(* IEC 61131-3 sources: ConveyorControl-with-PLC/4E_Gruppe1_Graf_Projekt1_HMI/Class/KeyPadAnum, 1 file *)

(* ---- KeyPadAnum.st ---- *)
(*!
<Class
	Name               = "KeyPadAnum"
	Revision           = "0.6"
	RealtimeTask       = "false"
	CyclicTask         = "false"
	BackgroundTask     = "false"
	Sigmatek           = "true"
	OSInterface        = "false"
	HighPriority       = "false"
	Automatic          = "false"
	UpdateMode         = "Prescan"
	IconPath           = ".\Class\KeyPadAnum\KeyPad.ico"
	SharedCommandTable = "true"
	Objectsize         = "(284,120)"
	Comment            = "class is used to get defaultimplementation of QWERTZ, QWERTY, AZERTY keyboard.&#13;&#10;keyboard differs on different languages&#13;&#10;set client &quot;Ima&quot; to IMA_WINDOW&#13;&#10;set client &quot;No&quot; to _WIN_EDITOR_ANUMERIC">
	<Channels>
		<Client Name="AltGr" Required="false" Internal="false" DefValue="1" Comment="set client to 1 when use of AltGr-key is necessary&#13;&#10;on the other hand client has to be set to 0"/>
		<Client Name="CapitalLetter" Required="false" Internal="false" DefValue="0" Comment="set client to 1 if capital letters are used without activated shift mode&#13;&#10;on the other hand set 0 to get capital letters when shift mode is activated"/>
		<Client Name="KeyPadImg" Required="true" Internal="true"/>
	</Channels>
	<RevDoku>
		<Owner Company="sigmatek" Author="kolott"/>
		<Dokumentation Revision="0.6" Date="2015-11-06" Author="kolott" Company="sigmatek" Description="sa32226, color of titlebar will work at several frames"/>
		<Dokumentation Revision="0.5" Date="2015-08-21" Author="kolott" Company="sigmatek" Description="betterment when using different frames"/>
		<Dokumentation Revision="0.4" Date="2014-02-07" Author="kolott" Company="sigmatek" Description="innovation titlelinepositioning"/>
		<Dokumentation Revision="0.3" Date="2013-10-02" Author="kolott" Company="sigmatek" Description="russian, ukrainian and greek keypad added"/>
		<Dokumentation Revision="0.1" Date="2013-07-10" Author="kolott" Company="sigmatek" Description="AltGr and CapitalLetter clients added"/>
		<Dokumentation Revision="0.0" Date="2013-03-06" Author="kolott" Company="sigmatek" Description="release"/>
	</RevDoku>
	<Network Name="KeyPadAnum">
		<!-- List of Components in this network -->
		<Components>
			<Object
				Name       = "_base"
				Class      = "_Screen"
				Position   = "(218,120)"
				Visualized = "true">
				<Channels>
					<Server Name="Screen"/>
					<Client Name="ImA" Value="IMA_WINDOW"/>
					<Client Name="Lse"/>
					<Client Name="No" Value="_WIN_EDITOR_ANUMERIC"/>
				</Channels>
			</Object>
			<Object
				Name       = "KeyPadImg"
				Class      = "KeyPadImages"
				Position   = "(210,420)"
				Visualized = "false">
				<Channels>
					<Server Name="ClassSvr"/>
				</Channels>
			</Object>
		</Components>
		<Comments>
		</Comments>
		<!-- List of Connections in this network -->
		<Connections>
			<Connection Source="this.Screen" Destination="_base.Screen" Vertices="(690,210),(518,210),"/>
			<Connection Source="_base.Lse" Destination="this.Lse" Vertices="(218,210),(38,210),"/>
			<Connection Source="_base.No" Destination="this.No" Vertices="(218,270),(38,270),"/>
			<Connection Source="_base.ImA" Destination="this.ImA" Vertices="(218,330),(38,330),"/>
			<Connection Source="this.KeyPadImg" Destination="KeyPadImg.ClassSvr"/>
		</Connections>
		<!-- Headerfiles -->
		<Options>
		</Options>
	</Network>
</Class>
*)
#pragma using _Screen

KeyPadAnum : CLASS
: _Screen
  //Servers:
  //Clients:
	KeyPadImg 	: CltChCmd_KeyPadImages;
	AltGr 	: CltCh_DINT;
	CapitalLetter 	: CltCh_DINT;
  //Variables:
		KeyButton_XOff 	: INT;
		KeyButton_YOff 	: INT;
		KeyButton_Width 	: INT;
		KeyButton_Height 	: INT;
		DoneByProgram 	: BOOL;
		YOff 	: INT;
  //Functions:

	FUNCTION KeyPadAnum
		VAR_OUTPUT
			ret_code 	: ConfStates;
		END_VAR;

	FUNCTION VIRTUAL GLOBAL S_Start
		VAR_INPUT
			pic 	: ^void;
			firsttime 	: BOOL;
		END_VAR;

	FUNCTION VIRTUAL GLOBAL S_CreateNew
		VAR_INPUT
			psetup 	: ^_NEWSCREENPROP;
		END_VAR
		VAR_OUTPUT
			retcode 	: BOOL;
		END_VAR;

	FUNCTION TAB KeyTab_QUERTZ;

	FUNCTION TAB KeyTab_QUERTY;

	FUNCTION VIRTUAL SelectKeyboard
		VAR_OUTPUT
			retcode 	: ^USINT;
		END_VAR;

	FUNCTION TAB KeyTab_FRENCH;

	FUNCTION TAB KeyTab_ITALIAN;

	FUNCTION TAB KeyTab_SPAIN;

	FUNCTION TAB KeyTab_PORTUGUESE;

	FUNCTION TAB KeyTab_NORWEGIAN;

	FUNCTION TAB KeyTab_SWEDISH;

	FUNCTION TAB SingleText;

	FUNCTION VIRTUAL GetBig
		VAR_INPUT
			pkey 	: ^USINT;
		END_VAR
		VAR_OUTPUT
			retcode 	: USINT;
		END_VAR;

	FUNCTION TAB KeyTab_CROATIAN_SERBIAN;

	FUNCTION TAB KeyTab_DANISH;

	FUNCTION TAB KeyTab_DUTCH;

	FUNCTION TAB KeyTab_RUSSIAN;

	FUNCTION IsUnicodeKeyboard
		VAR_INPUT
			pkey 	: ^USINT;
		END_VAR
		VAR_OUTPUT
			retcode 	: BOOL;
		END_VAR;

	FUNCTION TAB KeyTab_UKRAINIAN;

	FUNCTION TAB KeyTab_GREEK;
  //Tables:
	FUNCTION @STD
		VAR_OUTPUT
			ret_code	: CONFSTATES;
		END_VAR;
	FUNCTION GLOBAL TAB @CT_;
END_CLASS;

#pragma using KeyPadImages

FUNCTION TAB KeyPadAnum::SingleText

   0 , 0 , 0 , 0 , 0 , 0 , 0 , 0 , 0 , 0 , 0 , 0 , 0 , 0 , 0 , 0 , 0 , 0 , 0 , 0 , 0 , 0 , 0 , 0 , 0 , 0 , 0 , 0 , 0 , 0 , 0 , 0 , //   0- 31
   0 , 0 , 0 , 0 , 0 , 0 , 0 , 0 , 0 , 0 , 0 , 0 , 0 , 0 , 0 , 0 , 0 , 0 , 0 , 0 , 0 , 0 , 0 , 0 , 0 , 0 , 0 , 0 , 0 , 0 , 0 , 0 , //  32- 63
   0 ,'A','B','C','D','E','F','G','H','I','J','K','L','M','N','O','P','Q','R','S','T','U','V','W','X','Y','Z', 0 , 0 , 0 , 0 , 0 , //  64- 95
   0 ,'A','B','C','D','E','F','G','H','I','J','K','L','M','N','O','P','Q','R','S','T','U','V','W','X','Y','Z', 0 , 0 , 0 , 0 , 0 , //  96-127
   0 , 0 , 0 , 0 , 0 , 0 , 0 , 0 , 0 , 0 , 0 , 0 , 0 , 0 , 0 , 0 , 0 , 0 , 0 , 0 , 0 , 0 , 0 , 0 , 0 , 0 , 0 , 0 , 0 , 0 , 0 , 0 , // 128-159
   0 , 0 , 0 , 0 , 0 , 0 , 0 , 0 , 0 , 0 , 0 , 0 , 0 , 0 , 0 , 0 , 0 , 0 , 0 , 0 , 0 , 0 , 0 , 0 , 0 , 0 , 0 , 0 , 0 , 0 , 0 , 0 , // 160-191
   0 , 0 , 0 , 0 ,196,197,198,199, 0 , 0 , 0 , 0 , 0 , 0 , 0 , 0 , 0 ,209, 0 , 0 , 0 , 0 ,214, 0 ,216, 0 , 0 , 0 ,220, 0 , 0 , 0 , // 192-223
   0 , 0 , 0 , 0 ,196,197,198,199, 0 , 0 , 0 , 0 , 0 , 0 , 0 , 0 , 0 ,209, 0 , 0 , 0 , 0 ,214, 0 ,216, 0 , 0 , 0 ,220, 0 , 0 , 0 , // 224-255

END_FUNCTION

FUNCTION TAB KeyPadAnum::KeyTab_QUERTZ

  '1','!', 0 ,'2','"', 0 ,'3','§', 0 ,'4','$', 0 ,'5','%', 0 ,'6','&', 0 ,'7','/','{','8','(','[','9',')',']','0','=','}','ß','?','\',
  'q','Q','@','w','W', 0 ,'e','E', 0 ,'r','R', 0 ,'t','T', 0 ,'z','Z', 0 ,'u','U', 0 ,'i','I', 0 ,'o','O', 0 ,'p','P', 0 ,'ü','Ü', 0 ,
  'a','A', 0 ,'s','S', 0 ,'d','D', 0 ,'f','F', 0 ,'g','G', 0 ,'h','H', 0 ,'j','J', 0 ,'k','K', 0 ,'l','L', 0 ,'ö','Ö', 0 ,'ä','Ä', 0 ,
  'y','Y', 0 ,'x','X', 0 ,'c','C', 0 ,'v','V', 0 ,'b','B', 0 ,'n','N', 0 ,'m','M', 0 ,',',';', 0 ,'.',':', 0 ,'-','_', 0 ,'+','*', 0 ,

END_FUNCTION

FUNCTION TAB KeyPadAnum::KeyTab_QUERTY

  '1','!', 0 ,'2','@', 0 ,'3','#', 0 ,'4','$', 0 ,'5','%', 0 ,'6','^', 0 ,'7','&', 0 ,'8','*', 0 ,'9','(', 0 ,'0',')', 0 ,'=','+', 0 ,
  'q','Q', 0 ,'w','W', 0 ,'e','E', 0 ,'r','R', 0 ,'t','T', 0 ,'y','Y', 0 ,'u','U', 0 ,'i','I', 0 ,'o','O', 0 ,'p','P', 0 ,'[','{', 0 ,
  'a','A', 0 ,'s','S', 0 ,'d','D', 0 ,'f','F', 0 ,'g','G', 0 ,'h','H', 0 ,'j','J', 0 ,'k','K', 0 ,'l','L', 0 ,';',':', 0 ,']','}', 0 ,
  'z','Z', 0 ,'x','X', 0 ,'c','C', 0 ,'v','V', 0 ,'b','B', 0 ,'n','N', 0 ,'m','M', 0 ,',','<', 0 ,'.','>', 0 ,'/','?','\','-','_', 0 ,

END_FUNCTION

FUNCTION TAB KeyPadAnum::KeyTab_DUTCH

  '1','!','@','2','"', 0 ,'3','#', 0 ,'4','$', 0 ,'5','%', 0 ,'6','&', 0 ,'7','_', 0 ,'8','(','{','9',')','}','0',''', 0 ,'/','?','\',
  'q','Q', 0 ,'w','W', 0 ,'e','E', 0 ,'r','R', 0 ,'t','T', 0 ,'y','Y', 0 ,'u','U', 0 ,'i','I', 0 ,'o','O', 0 ,'p','P', 0 ,'*','°', 0 ,
  'a','A', 0 ,'s','S','ß','d','D', 0 ,'f','F', 0 ,'g','G', 0 ,'h','H', 0 ,'j','J', 0 ,'k','K', 0 ,'l','L', 0 ,'+',177, 0 ,'<','>', 0 ,
  'z','Z', 0 ,'x','X', 0 ,'c','C', 0 ,'v','V', 0 ,'b','B', 0 ,'n','N', 0 ,'m','M', 0 ,',',';', 0 ,'.',':', 0 ,'-','=', 0 ,'[',']', 0 ,

END_FUNCTION

FUNCTION TAB KeyPadAnum::KeyTab_FRENCH

  '&','1', 0 ,233,'2','~','"','3','#',''','4','{','(','5','[','-','6', 0 ,232,'7', 0 ,'_','8','\',231,'9','^',224,'0','@',')','°',']',
  'a','A', 0 ,'z','Z', 0 ,'e','E', 0 ,'r','R', 0 ,'t','T', 0 ,'y','Y', 0 ,'u','U', 0 ,'i','I', 0 ,'o','O', 0 ,'p','P', 0 ,'=','+','}',
  'q','Q', 0 ,'s','S', 0 ,'d','D', 0 ,'f','F', 0 ,'g','G', 0 ,'h','H', 0 ,'j','J', 0 ,'k','K', 0 ,'l','L', 0 ,'m','M', 0 ,249,'%', 0 ,
  'w','W', 0 ,'x','X', 0 ,'c','C', 0 ,'v','V', 0 ,'b','B', 0 ,'n','N', 0 ,',','?', 0 ,';','.', 0 ,':','/', 0 ,'!','§', 0 ,'<','>', 0 ,

END_FUNCTION

FUNCTION TAB KeyPadAnum::KeyTab_ITALIAN

  '1','!', 0 ,'2','"', 0 ,'3',163, 0 ,'4','$', 0 ,'5','%', 0 ,'6','&', 0 ,'7','/','{','8','(','[','9',')',']','0','=','}','+','*', 0 ,
  'q','Q', 0 ,'w','W', 0 ,'e','E', 0 ,'r','R', 0 ,'t','T', 0 ,'y','Y', 0 ,'u','U', 0 ,'i','I', 0 ,'o','O', 0 ,'p','P', 0 ,232,233, 0 ,
  'a','A', 0 ,'s','S', 0 ,'d','D', 0 ,'f','F', 0 ,'g','G', 0 ,'h','H', 0 ,'j','J', 0 ,'k','K', 0 ,'l','L', 0 ,242,231,'@',224,'°','#',
  'z','Z', 0 ,'x','X', 0 ,'c','C', 0 ,'v','V', 0 ,'b','B', 0 ,'n','N', 0 ,'m','M', 0 ,',',';', 0 ,'.',':', 0 ,'-','_', 0 ,'<','>', 0 ,

END_FUNCTION

FUNCTION TAB KeyPadAnum::KeyTab_SPAIN

  '1','!','\','2','"','@','3','.','#','4','$','~','5','%', 0 ,'6','&', 0 ,'7','/','{','8','(','[','9',')',']','0','=','}',''','?', 0 ,
  'q','Q', 0 ,'w','W', 0 ,'e','E', 0 ,'r','R', 0 ,'t','T', 0 ,'y','Y', 0 ,'u','U', 0 ,'i','I', 0 ,'o','O', 0 ,'p','P', 0 ,'+','*', 0 ,
  'a','A', 0 ,'s','S', 0 ,'d','D', 0 ,'f','F', 0 ,'g','G', 0 ,'h','H', 0 ,'j','J', 0 ,'k','K', 0 ,'l','L', 0 ,241,209, 0 ,231,199, 0 ,
  'z','Z', 0 ,'x','X', 0 ,'c','C', 0 ,'v','V', 0 ,'b','B', 0 ,'n','N', 0 ,'m','M', 0 ,',',';', 0 ,'.',':', 0 ,'-','_', 0 ,'<','>', 0 ,

END_FUNCTION

FUNCTION TAB KeyPadAnum::KeyTab_PORTUGUESE

  '1','!', 0 ,'2','@', 0 ,'3','#', 0 ,'4','$', 0 ,'5','%', 0 ,'6','"', 0 ,'7','&', 0 ,'8','*', 0 ,'9','(','{','0',')','}','-','_', 0 ,
  'q','Q','/','w','W', 0 ,'e','E', 0 ,'r','R', 0 ,'t','T', 0 ,'y','Y', 0 ,'u','U', 0 ,'i','I', 0 ,'o','O', 0 ,'p','P', 0 ,'+','=','§',
  'a','A', 0 ,'s','S', 0 ,'d','D', 0 ,'f','F', 0 ,'g','G', 0 ,'h','H', 0 ,'j','J', 0 ,'k','K', 0 ,'l','L', 0 ,231,199, 0 ,'[',']','~',
  'z','Z', 0 ,'x','X', 0 ,'c','C', 0 ,'v','V', 0 ,'b','B', 0 ,'n','N', 0 ,'m','M', 0 ,',','<', 0 ,'.','>', 0 ,';',':', 0 ,'/','?', 0 ,

END_FUNCTION

FUNCTION TAB KeyPadAnum::KeyTab_NORWEGIAN

  '1','!', 0 ,'2','"','@','3','#', 0 ,'4',164,'$','5','%', 0 ,'6','&', 0 ,'7','/','{','8','(','[','9',')',']','0','=','}','+','?', 0 ,
  'q','Q', 0 ,'w','W', 0 ,'e','E', 0 ,'r','R', 0 ,'t','T', 0 ,'y','Y', 0 ,'u','U', 0 ,'i','I', 0 ,'o','O', 0 ,'p','P', 0 ,229,197, 0 ,
  'a','A', 0 ,'s','S', 0 ,'d','D', 0 ,'f','F', 0 ,'g','G', 0 ,'h','H', 0 ,'j','J', 0 ,'k','K', 0 ,'l','L', 0 ,248,216, 0 ,230,198, 0 ,
  'z','Z', 0 ,'x','X', 0 ,'c','C', 0 ,'v','V', 0 ,'b','B', 0 ,'n','N', 0 ,'m','M', 0 ,',',';', 0 ,'.',':', 0 ,'-','_', 0 ,'\','*', 0 ,

END_FUNCTION

FUNCTION TAB KeyPadAnum::KeyTab_DANISH

  '1','!', 0 ,'2','"','@','3','#', 0 ,'4',164,'$','5','%', 0 ,'6','&', 0 ,'7','/','{','8','(','[','9',')',']','0','=','}','+','?', 0 ,
  'q','Q', 0 ,'w','W', 0 ,'e','E', 0 ,'r','R', 0 ,'t','T', 0 ,'y','Y', 0 ,'u','U', 0 ,'i','I', 0 ,'o','O', 0 ,'p','P', 0 ,229,197, 0 ,
  'a','A', 0 ,'s','S', 0 ,'d','D', 0 ,'f','F', 0 ,'g','G', 0 ,'h','H', 0 ,'j','J', 0 ,'k','K', 0 ,'l','L', 0 ,230,198, 0 ,248,216, 0 ,
  'z','Z', 0 ,'x','X', 0 ,'c','C', 0 ,'v','V', 0 ,'b','B', 0 ,'n','N', 0 ,'m','M', 0 ,',',';', 0 ,'.',':', 0 ,'-','_', 0 ,'\','*', 0 ,

END_FUNCTION

FUNCTION TAB KeyPadAnum::KeyTab_SWEDISH

  '1','!', 0 ,'2','"','@','3','#', 0 ,'4',164,'$','5','%', 0 ,'6','&', 0 ,'7','/','{','8','(','[','9',')',']','0','=','}','+','?','\',
  'q','Q', 0 ,'w','W', 0 ,'e','E', 0 ,'r','R', 0 ,'t','T', 0 ,'y','Y', 0 ,'u','U', 0 ,'i','I', 0 ,'o','O', 0 ,'p','P', 0 ,229,197, 0 ,
  'a','A', 0 ,'s','S', 0 ,'d','D', 0 ,'f','F', 0 ,'g','G', 0 ,'h','H', 0 ,'j','J', 0 ,'k','K', 0 ,'l','L', 0 ,'ö','Ö', 0 ,'ä','Ä', 0 ,
  'z','Z', 0 ,'x','X', 0 ,'c','C', 0 ,'v','V', 0 ,'b','B', 0 ,'n','N', 0 ,'m','M', 0 ,',',';', 0 ,'.',':', 0 ,'-','_', 0 ,'~','*', 0 ,

END_FUNCTION

FUNCTION TAB KeyPadAnum::KeyTab_RUSSIAN

    49$uint,  33$uint,  0$uint,    50$uint,  34$uint,  0$uint,    51$uint,  21$uint,  0$uint,    52$uint,  59$uint,  0$uint,    53$uint,  37$uint,  0$uint,
    54$uint,  58$uint,  0$uint,    55$uint,  63$uint,  0$uint,    56$uint,  42$uint,  0$uint,    57$uint,  40$uint,  0$uint,    48$uint,  41$uint,  0$uint,    45$uint,  95$uint,0$uint,
  1081$uint,1049$uint,'Q'$uint,  1094$uint,1062$uint,'W'$uint,  1091$uint,1059$uint,'E'$uint,  1082$uint,1050$uint,'R'$uint,  1077$uint,1045$uint,'T'$uint,
  1085$uint,1053$uint,'Y'$uint,  1075$uint,1043$uint,'U'$uint,  1096$uint,1064$uint,'I'$uint,  1097$uint,1065$uint,'O'$uint,  1079$uint,1047$uint,'P'$uint,  1093$uint,1061$uint,0$uint,
  1092$uint,1060$uint,'A'$uint,  1099$uint,1067$uint,'S'$uint,  1074$uint,1042$uint,'D'$uint,  1072$uint,1040$uint,'F'$uint,  1087$uint,1055$uint,'G'$uint,
  1088$uint,1056$uint,'H'$uint,  1086$uint,1054$uint,'J'$uint,  1083$uint,1051$uint,'K'$uint,  1076$uint,1044$uint,'L'$uint,  1078$uint,1046$uint,  0$uint,  1101$uint,1069$uint,0$uint,
  1103$uint,1071$uint,'Z'$uint,  1095$uint,1063$uint,'X'$uint,  1089$uint,1057$uint,'C'$uint,  1084$uint,1052$uint,'V'$uint,  1080$uint,1048$uint,'B'$uint,
  1090$uint,1058$uint,'N'$uint,  1100$uint,1068$uint,'M'$uint,  1073$uint,1041$uint,  0$uint,  1102$uint,1070$uint,  0$uint,  1098$uint,1066$uint,  0$uint,    46$uint,  44$uint,0$uint

END_FUNCTION

FUNCTION TAB KeyPadAnum::KeyTab_UKRAINIAN

    49$uint,  33$uint,  0$uint,   50$uint,  34$uint,  0$uint,   51$uint,  21$uint,  0$uint,   52$uint,  59$uint,  0$uint,   53$uint,  37$uint,  0$uint,
    54$uint,  58$uint,  0$uint,   55$uint,  63$uint,  0$uint,   56$uint,  42$uint,  0$uint,   57$uint,  40$uint,  0$uint,   48$uint,  41$uint,  0$uint,   45$uint,  95$uint,0$uint,
  1081$uint,1049$uint,'Q'$uint, 1094$uint,1062$uint,'W'$uint, 1091$uint,1059$uint,'E'$uint, 1082$uint,1050$uint,'R'$uint, 1077$uint,1045$uint,'T'$uint,
  1085$uint,1053$uint,'Y'$uint, 1075$uint,1043$uint,'U'$uint, 1096$uint,1064$uint,'I'$uint, 1097$uint,1065$uint,'O'$uint, 1079$uint,1047$uint,'P'$uint, 1093$uint,1061$uint,0$uint,
  1092$uint,1060$uint,'A'$uint, 1110$uint,1030$uint,'S'$uint, 1074$uint,1042$uint,'D'$uint, 1072$uint,1040$uint,'F'$uint, 1087$uint,1055$uint,'G'$uint,
  1088$uint,1056$uint,'H'$uint, 1086$uint,1054$uint,'J'$uint, 1083$uint,1051$uint,'K'$uint, 1076$uint,1044$uint,'L'$uint, 1078$uint,1046$uint,  0$uint, 1108$uint,1028$uint,0$uint,
  1103$uint,1071$uint,'Z'$uint, 1095$uint,1063$uint,'X'$uint, 1089$uint,1057$uint,'C'$uint, 1084$uint,1052$uint,'V'$uint, 1080$uint,1048$uint,'B'$uint,
  1090$uint,1058$uint,'N'$uint, 1100$uint,1068$uint,'M'$uint, 1073$uint,1041$uint,  0$uint, 1102$uint,1070$uint,  0$uint, 1111$uint,1031$uint,  0$uint,   46$uint,  44$uint,0$uint

END_FUNCTION

FUNCTION TAB KeyPadAnum::KeyTab_GREEK

  '1'$uint,'!'$uint,  0$uint,  '2'$uint,'@'$uint,  0$uint, '3'$uint,'#'$uint,  0$uint, '4'$uint,'$'$uint,  0$uint, '5'$uint,'%'$uint,  0$uint,
  '6'$uint,'^'$uint,  0$uint,  '7'$uint,'&'$uint,  0$uint, '8'$uint,'*'$uint,  0$uint, '9'$uint,'('$uint,  0$uint, '0'$uint,')'$uint,  0$uint, '-'$uint, '_'$uint,0$uint,
  ';'$uint,':'$uint,'Q'$uint,  962$uint,962$uint,'W'$uint, 949$uint,917$uint,'E'$uint, 961$uint,929$uint,'R'$uint, 964$uint,932$uint,'T'$uint,
  965$uint,933$uint,'Y'$uint,  952$uint,920$uint,'U'$uint, 953$uint,921$uint,'I'$uint, 959$uint,927$uint,'O'$uint, 960$uint,928$uint,'P'$uint, '{'$uint,'['$uint,0$uint,
  945$uint,913$uint,'A'$uint,  963$uint,931$uint,'S'$uint, 948$uint,916$uint,'D'$uint, 966$uint,934$uint,'F'$uint, 947$uint,915$uint,'G'$uint,
  951$uint,919$uint,'H'$uint,  958$uint,926$uint,'J'$uint, 954$uint,922$uint,'K'$uint, 955$uint,923$uint,'L'$uint,  39$uint,'"'$uint,  0$uint, '}'$uint,']'$uint,0$uint,
  950$uint,918$uint,'Z'$uint,  967$uint,935$uint,'X'$uint, 968$uint,936$uint,'C'$uint, 969$uint,937$uint,'V'$uint, 946$uint,914$uint,'B'$uint,
  957$uint,925$uint,'N'$uint,  956$uint,924$uint,'M'$uint, '<'$uint,','$uint,  0$uint, '>'$uint,'.'$uint,  0$uint, '?'$uint,'/'$uint,  0$uint, '+'$uint,'='$uint,0$uint

END_FUNCTION

FUNCTION VIRTUAL KeyPadAnum::SelectKeyboard
	VAR_OUTPUT
		retcode 	: ^USINT;
	END_VAR

  retcode := #KeyTab_QUERTY()$^usint;
  case Language_GetActualLocal() of
    LOCAL_GERMAN    : retcode := #KeyTab_QUERTZ()$^usint;
    LOCAL_DUTCH     : retcode := #KeyTab_DUTCH()$^usint;
    LOCAL_FRENCH    : retcode := #KeyTab_FRENCH()$^usint;
    LOCAL_ITALIAN   : retcode := #KeyTab_ITALIAN()$^usint;
    LOCAL_SPANISH   : retcode := #KeyTab_SPAIN()$^usint;
    LOCAL_PORTUGESE : retcode := #KeyTab_PORTUGUESE()$^usint;
    LOCAL_NORWEGIAN : retcode := #KeyTab_NORWEGIAN()$^usint;
    LOCAL_FINNISH,
    LOCAL_SWEDISH   : retcode := #KeyTab_SWEDISH()$^usint;
    LOCAL_DANISH    : retcode := #KeyTab_DANISH()$^usint;
    LOCAL_UKRAINIAN : retcode := #KeyTab_UKRAINIAN()$^usint;
    LOCAL_RUSSIAN   : retcode := #KeyTab_RUSSIAN()$^usint;
    LOCAL_GREEK     : retcode := #KeyTab_GREEK()$^usint;
  end_case;

  retcode += 4;

END_FUNCTION

FUNCTION KeyPadAnum::IsUnicodeKeyboard
	VAR_INPUT
		pkey 	: ^USINT;
	END_VAR
	VAR_OUTPUT
		retcode 	: BOOL;
	END_VAR
  VAR
  	pukbrd : ^udint;
  END_VAR

  retcode := false;
  pukbrd  := #KeyTab_RUSSIAN();
  pkey    -= 4;
  if(pkey$^udint^ = pukbrd^) then
    retcode := true;
  end_if;

END_FUNCTION

FUNCTION KeyPadAnum::KeyPadAnum
	VAR_OUTPUT
		ret_code 	: ConfStates;
	END_VAR

	ret_code         := C_OK;
  KeyButton_XOff   := 5;
  KeyButton_YOff   := 37;
  KeyButton_Width  := 50;
  KeyButton_Height := 50;

END_FUNCTION

FUNCTION VIRTUAL GLOBAL KeyPadAnum::S_CreateNew
	VAR_INPUT
		psetup 	: ^_NEWSCREENPROP;
	END_VAR
	VAR_OUTPUT
		retcode 	: BOOL;
	END_VAR
  VAR
  	room : _ROOM;
    tmp, xx, yy : int;
    pdkp : ^_DEFKEYPAD;
  END_VAR

  retcode       := true;
  DoneByProgram := true;

  MyGetScreenSize(#room);
  xx := 640; // keypad width
  yy := 342; // keypad height

  //room.xy2.x := 479; // test small display
  if(room.xy2.x < 639) then
    KeyButton_XOff   := 4;
    KeyButton_Width  := 37;
    KeyButton_Height := 44; // 37
    xx               := 480;
    yy               := 304; // 265
  end_if;

  pdkp := Get_DEFKEYPAD();
  tmp  := KeyPadImg.GetTitleLineHeight(pdkp^.WindowFrame) - KeyPadImg.GetTitleLineHeight(FRAME_NONE);
  YOff := KeyButton_YOff + tmp;
  yy   += tmp;

  psetup^.Position.xy1.x     := (room.xy2.x - room.xy1.x + 1 - xx) / 2;
  psetup^.Position.xy1.y     := (room.xy2.y - room.xy1.y + 1 - yy) / 2;
  psetup^.Position.xy2.x     := psetup^.Position.xy1.x + xx - 1;
  psetup^.Position.xy2.y     := psetup^.Position.xy1.y + yy - 1;
  psetup^.FrameId            := pdkp^.WindowFrame;
  psetup^.TouchEditorAscii   := false;
  psetup^.TouchEditorNumeric := false;
  psetup^.ColorBack          := pdkp^.WindowColorBack;
  psetup^.ColorHatch         := pdkp^.TitleBarColor;  // sa32226

END_FUNCTION

FUNCTION VIRTUAL KeyPadAnum::GetBig
	VAR_INPUT
		pkey 	: ^USINT;
	END_VAR
	VAR_OUTPUT
		retcode 	: USINT;
	END_VAR
  VAR
  	pc1, pc2 : ^usint;
  END_VAR

  retcode := 0;
  pc1  := #SingleText()$^usint + 4 + pkey^; pkey += 1;
  pc2  := #SingleText()$^usint + 4 + pkey^;
  if(pc1^= pc2^) then
    retcode := pc1^;
  end_if;

END_FUNCTION

FUNCTION VIRTUAL GLOBAL KeyPadAnum::S_Start
	VAR_INPUT
		pic 	: ^void;
		firsttime 	: BOOL;
	END_VAR
  VAR
    room : _ROOM;
  	style, stylegr : _STYLESHEET;
    x, y : _KOORD;
    any : _ANYPARA;
    pkey : ^usint;
    big : usint;
    code : array[0..2] of usint;
    ucode : array[0..2] of uint;
    str : array[0..5] of char;
    ustr : array[0..5] of uint;
    ino, jno : udint;
    pdkp : ^_DEFKEYPAD;
  END_VAR

  if(DoneByProgram = true) & (firsttime = true) then

    CapitalLetter := CapitalLetter.Read();
    AltGr         := AltGr.Read();
    pdkp          := Get_DEFKEYPAD();

    init_STYLESHEET(#style);
    setup_STYLESHEET(#style, #pdkp^.StandardFontSchemeName[0], pdkp^.ButtonFrame, T_CENTERBOUND or T_MIDBOUND, pdkp^.ButtonColorReleased, pdkp^.ButtonColorText, pdkp^.ButtonColorPressed, WHITE, DARKGRAY, NIL, NIL, NIL, NIL, NIL);

    pkey := SelectKeyboard();
    if(IsUnicodeKeyboard(pkey) = true) then
      for y:=0 to 3 do
        for x:=0 to 10 do
          room.xy1.x := Keybutton_XOff + y * 10 + x * KeyButton_Width;
          room.xy1.y := YOff + y * KeyButton_Height + KeyButton_Height;
          room.xy2.x := room.xy1.x + (KeyButton_Width - 2);
          room.xy2.y := room.xy1.y + (KeyButton_Height - 2);

          ucode[0]  := pkey$^uint^; pkey += 2;
          ucode[1]  := pkey$^uint^; pkey += 2;
          ucode[2]  := _NOKEY;
          if(AltGr = 1) then
            ucode[2] := pkey$^uint^;
          end_if;
          pkey += 2;

          if(((ucode[0] - ucode[1]) = 32) | (ucode[0] = ucode[1])) then
            ustr[0] := ucode[1];
            ustr[1] := 0;

            if(CapitalLetter = 1) then
              ustr[0]  := ucode[0] ;
              ucode[0] := ucode[1];
              ucode[1] := ustr[0];
            end_if;
          else
            ustr[0] := ucode[1];
            ustr[1] := '|';
            ustr[2] := ucode[0];
            ustr[3] := 0;
          end_if;

          add_key(pic$^_MY_PICTURE, #style, #room, DEFSCOPE, #ustr[0], sizeof(_UNI), T_CENTERBOUND or T_MIDBOUND, ucode[0], ucode[1], ucode[2]);
        end_for;
      end_for;
    else
      for y:=0 to 3 do
        for x:=0 to 10 do
          room.xy1.x := Keybutton_XOff + y * 10 + x * KeyButton_Width;
          room.xy1.y := YOff + y * KeyButton_Height + KeyButton_Height;
          room.xy2.x := room.xy1.x + (KeyButton_Width - 2);
          room.xy2.y := room.xy1.y + (KeyButton_Height - 2);

          code$uint := pkey$^uint^;
          code[2]   := _NOKEY;
          if(AltGr = 1) then
            code[2] := (pkey+2)^;
          end_if;

          big := GetBig(pkey);
          if(big <> 0) then
            str[0] := big;
            str[1] := 0;

            if(CapitalLetter = 1) then
              str[0]  := str[0] xor ('a' xor 'A');
              code[0] := code[1];
              code[1] := pkey^;
            end_if;
          else
            str[0] := (pkey + 1)^;
            str[1] := '|';
            str[2] := pkey^;
            str[3] := 0;
          end_if;

          add_key(pic$^_MY_PICTURE, #style, #room, DEFSCOPE, #str[0], sizeof(_ASCII), T_CENTERBOUND or T_MIDBOUND, code[0], code[1], code[2]);
          pkey += 3;
        end_for;
      end_for;
    end_if;

    // key backspace
    room.xy1.x := Keybutton_XOff + 10 + KeyButton_Width * 11;
    room.xy1.y := YOff + KeyButton_Height;
    room.xy2.x := room.xy1.x + (KeyButton_Width + 20 - 2);
    room.xy2.y := room.xy1.y + (KeyButton_Height - 2);
    ino := KeyPadImg.GetImage(0);
    add_key(pic$^_MY_PICTURE, #style, #room, ino, NIL, sizeof(_ASCII), T_CENTERBOUND or T_MIDBOUND, _BCKSPC, _BCKSPC);

    // key insert
    room.xy1.x := room.xy2.x - (KeyButton_Width - 2);
    room.xy1.y := room.xy2.y + 2;
    room.xy2.y := room.xy1.y + (KeyButton_Height - 2);
    add_button(pic$^_MY_PICTURE, #style, #room, DEFSCOPE, DEFSCOPE, DEFSCOPE, VARNO_INSERTFLAG, DEFSCOPE, DEFSCOPE, "Ins", "Ins", sizeof(_ASCII), false, 0, 0, DEFSCOPE, 1, 0, T_CENTERBOUND or T_MIDBOUND);

    // key enter
    room.xy1.y := room.xy2.y + 2;
    room.xy2.y := room.xy1.y + (2 * KeyButton_Height - 2);
    ino := KeyPadImg.GetImage(1);
    //add_button(pic$^_MY_PICTURE, #style, #room, DEFSCOPE, DEFSCOPE, DEFSCOPE, DEFSCOPE, ino, ino, NIL, NIL, sizeof(_ASCII), true, 0, 0, DEFSCOPE, 1, 0, T_CENTERBOUND or T_MIDBOUND);
    add_key(pic$^_MY_PICTURE, #style, #room, ino, NIL, sizeof(_ASCII), T_CENTERBOUND or T_MIDBOUND, _ENTER, _ENTER);

    // key right
    room.xy1.y := room.xy2.y + 2;
    room.xy2.y := room.xy1.y + KeyButton_Height - 2;
    ino := KeyPadImg.GetImage(2);
    add_key(pic$^_MY_PICTURE, #style, #room, ino, NIL, sizeof(_ASCII), T_CENTERBOUND or T_MIDBOUND, _RIGHT, _RIGHT);

    // key left
    room.xy1.x := room.xy1.x - KeyButton_Width;
    room.xy2.x := room.xy2.x - KeyButton_Width;
    ino := KeyPadImg.GetImage(3);
    add_key(pic$^_MY_PICTURE, #style, #room, ino, NIL, sizeof(_ASCII), T_CENTERBOUND or T_MIDBOUND, _LEFT, _LEFT);

    ino := 5;
    jno := 4;
    if(CapitalLetter = 1) then
      ino := 4;
      jno := 5;
    end_if;
    ino := KeyPadImg.GetImage(ino);
    jno := KeyPadImg.GetImage(jno);
    if(AltGr = 0) then
      // key shift (right)
      room.xy2.x := room.xy1.x - 2;
      room.xy1.x := room.xy2.x - (KeyButton_Width + 20 - 2);
      add_button(pic$^_MY_PICTURE, #style, #room, DEFSCOPE, DEFSCOPE, DEFSCOPE, VARNO_SHIFTFLAG, ino, jno, NIL, NIL, sizeof(_ASCII), false, 0, 0, DEFSCOPE, 1, 0, T_CENTERBOUND or T_MIDBOUND);
    else
      // key altgr (right)
      init_STYLESHEET(#stylegr);
      setup_STYLESHEET(#stylegr, #pdkp^.StandardFontSchemeName[0], pdkp^.ButtonFrame, T_CENTERBOUND or T_MIDBOUND, pdkp^.ButtonColorReleased, pdkp^.ButtonColorText, LIGHTCYAN, WHITE, DARKGRAY, NIL, NIL, NIL, NIL, NIL);
      room.xy2.x := room.xy1.x - 2;
      room.xy1.x := room.xy2.x - (KeyButton_Width + 20 - 2);
      add_button(pic$^_MY_PICTURE, #stylegr, #room, DEFSCOPE, DEFSCOPE, DEFSCOPE, VARNO_ALTGRFLAG, DEFSCOPE, DEFSCOPE, "AltGr", "AltGr", sizeof(_ASCII), false, 0, 0, DEFSCOPE, 1, 0, T_CENTERBOUND or T_MIDBOUND);
      free_STYLESHEET(#stylegr);
    end_if;

    // key shift (left)
    room.xy1.x := Keybutton_XOff;
    room.xy2.x := room.xy1.x + (KeyButton_Width + 20 - 2);
    add_button(pic$^_MY_PICTURE, #style, #room, DEFSCOPE, DEFSCOPE, DEFSCOPE, VARNO_SHIFTFLAG, ino, jno, NIL, NIL, sizeof(_ASCII), false, 0, 0, DEFSCOPE, 1, 0, T_CENTERBOUND or T_MIDBOUND);

    // key space
    room.xy1.x := Keybutton_XOff + (KeyButton_Width + 20);
    room.xy2.x := Keybutton_XOff + 9 * KeyButton_Width - 2 + 10;
    add_key(pic$^_MY_PICTURE, #style, #room, DEFSCOPE, NIL, sizeof(_ASCII), T_CENTERBOUND or T_MIDBOUND, ' ', ' ');

    // input
    setup_STYLESHEET(#style, #pdkp^.StandardFontSchemeName[0], FRAME_STEALTH, T_CENTERBOUND or T_MIDBOUND or T_INVERTTHEME, LIGHTGRAY, WHITE, LIGHTGRAY, WHITE, DARKGRAY, NIL, NIL, NIL, NIL, NIL);
    room.xy1.x := Keybutton_XOff;
    room.xy1.y := YOff;
    room.xy2.x := room.xy1.x + 10 + (KeyButton_Width * 12 + 20 - 2);
    room.xy2.y := room.xy1.y + KeyButton_Height - 6;
    add_input(pic$^_MY_PICTURE, #style, #room, DEFSCOPE, VARNO_EDITORDUMMY, AS_ASCII, DEFSCOPE);

    // titletext
    if(pdkp^.TitleColorText$UINT <> INVISIBLE) then
      setup_STYLESHEET(#style, #pdkp^.StandardFontSchemeName[0], FRAME_NONE, T_LEFTBOUND or T_MIDBOUND, INVISIBLE, pdkp^.TitleColorText, INVISIBLE, INVISIBLE, INVISIBLE, NIL, NIL, NIL, NIL, NIL);
      room.xy1.x := Keybutton_XOff;
      room.xy1.y := 2;
      room.xy2.x := room.xy1.x + (KeyButton_Width * 12); //400;
      room.xy2.y := 2 + KeyPadImg.GetTitleLineHeight(pdkp^.WindowFrame);
      init_ANYPARA(#any);
      any.anything.list := VARTXT1;
      any.anything.no   := VARNO_EDITORDUMMY;
      add_text(pic$^_MY_PICTURE, #style, #room, DEFSCOPE, #any, NIL, sizeof(_ASCII), DEFSCOPE);
    end_if;

    if(has_theme_cancel(pdkp^.WindowFrame) = false) then
      // cancel button
      setup_STYLESHEET(#style, #pdkp^.StandardFontSchemeName[0], pdkp^.ButtonFrame, T_CENTERBOUND or T_MIDBOUND, 16#F800, pdkp^.ButtonColorText, RED, WHITE, DARKGRAY, NIL, NIL, NIL, NIL, NIL);
      room.xy1.x := Keybutton_XOff + (KeyButton_Width * 12) + 2;
      room.xy1.y := 5;
      room.xy2.x := room.xy1.x + 26;
      room.xy2.y := 31;
      ino := KeyPadImg.GetImage(6);
      add_key(pic$^_MY_PICTURE, #style, #room, ino, NIL, sizeof(_ASCII), T_CENTERBOUND or T_MIDBOUND, _ESC, _ESC);
    end_if;

    free_ANYPARA(#any);
    free_STYLESHEET(#style);
  end_if;

END_FUNCTION
